TYPE ST_MotionlinxAI_Axis_Command :
	STRUCT
		Extend	: BOOL;
		Retract : BOOL;
	END_STRUCT
END_TYPE

(* stored: Version 1.1.0.1, ProductVersion 3.1.4024.15
   DUT ST_MotionlinxAI_Axis_Command: Id {cd4d3ba9-cab6-4bd6-959d-da15cd2042c9} *)
